FUNCTION LogMessage : DINT
VAR_INPUT
	msg		: STRING;
	hSocket	: T_HSOCKET;
END_VAR
VAR
END_VAR

IF bLogDebugMessages THEN
	LogMessage := ADSLOGDINT( ADSLOG_MSGTYPE_HINT OR ADSLOG_MSGTYPE_LOG, CONCAT( msg, '::Internal handle: %d' ), UDINT_TO_DINT(hSocket.handle)  );
END_IF

END_FUNCTION

(* stored: Version 1.1.0.1, ProductVersion 3.1.4024.12
   POU LogMessage: Id {ee3bdd69-1a87-4b05-ac8e-db0bceeacd9c}, SpecialFunc None *)
